{attribute 'GeneratedUsingTerminal: EK1122-0000-0018'}
{attribute addProperty BoxType "EK1122-0000-0018"}
{attribute addProperty Id "Beckhoff_EM3xxxsub_EK1100EK1100_1FC0878B2"}
{attribute addProperty CRC "4277636301"}
{attribute addProperty Size "2"}
TYPE Beckhoff_EM3xxxEK1122_FEF78CCD EXTENDS EK1122_1FC0878B :
STRUCT
	{attribute addProperty Name "Beckhoff EM3xxxsub EK1100"}
	{attribute addProperty PreviousPort "Beckhoff EM3xxxEK1122 : D"}
	Beckhoff_EM3xxxsub_EK1100 : EK1100_1FC0878B;
END_STRUCT
END_TYPE
